Staubli VAL3: ToolItem.dtx

public InstrItem iActionOFF[3]
  [0]
    string sType
    string sData
  [1]
    string sType
    string sData
  [2]
    string sType
    string sData
public InstrItem iActionON[3]
  [0]
    string sType
    string sData
  [1]
    string sType
    string sData
  [2]
    string sType
    string sData
public string name
public tool tcp = {fatherId=flange[0], ioLink=valve1}
